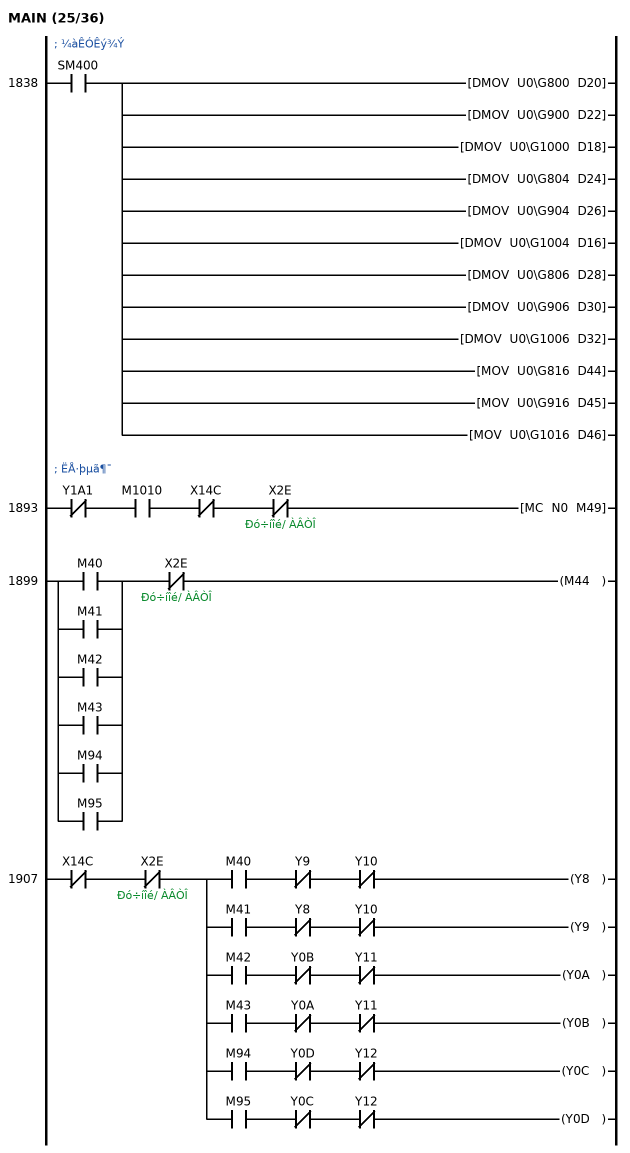
[picture p24: ladder of MAIN, rungs at steps 1838 to 1907]
; 监视数据
1838  LD      SM400
      DMOV    U0\G800 D20
      DMOV    U0\G900 D22
      DMOV    U0\G1000 D18
      DMOV    U0\G804 D24
      DMOV    U0\G904 D26
      DMOV    U0\G1004 D16
      DMOV    U0\G806 D28
      DMOV    U0\G906 D30
      DMOV    U0\G1006 D32
      MOV     U0\G816 D44
      MOV     U0\G916 D45
      MOV     U0\G1016 D46
; 伺服点动
1893  LDI     Y1A1
      AND     M1010
      ANI     X14C
      ANI     X2E  ; Ручной/ АВТО
      MC      N0 M49
1899  LD      M40
      OR      M41
      OR      M42
      OR      M43
      OR      M94
      OR      M95
      ANI     X2E  ; Ручной/ АВТО
      OUT     M44
1907  LDI     X14C
      ANI     X2E  ; Ручной/ АВТО
      MPS
      AND     M40
      ANI     Y9
      ANI     Y10
      OUT     Y8
      MRD
      AND     M41
      ANI     Y8
      ANI     Y10
      OUT     Y9
      MRD
      AND     M42
      ANI     Y0B
      ANI     Y11
      OUT     Y0A
      MRD
      AND     M43
      ANI     Y0A
      ANI     Y11
      OUT     Y0B
      MRD
      AND     M94
      ANI     Y0D
      ANI     Y12
      OUT     Y0C
      MPP
      AND     M95
      ANI     Y0C
      ANI     Y12
      OUT     Y0D
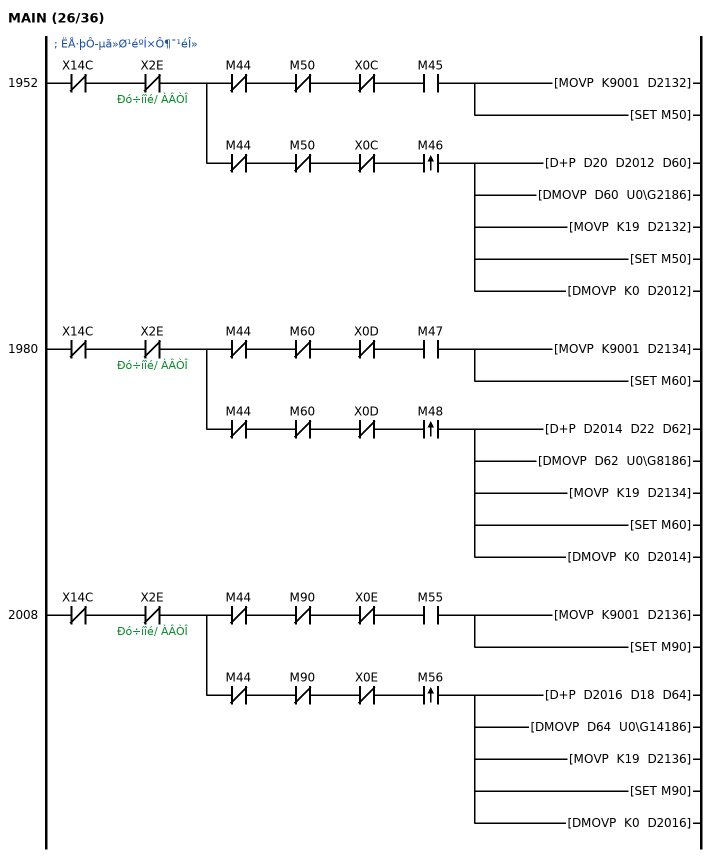
; 伺服原点回归和自动归位
1952  LDI     X14C
      ANI     X2E  ; Ручной/ АВТО
      MPS
      ANI     M44
      ANI     M50
      ANI     X0C
      AND     M45
      MOVP    K9001 D2132
      SET     M50
      MPP
      ANI     M44
      ANI     M50
      ANI     X0C
      ANDP    M46
      D+P     D20 D2012 D60
      DMOVP   D60 U0\G2186
      MOVP    K19 D2132
      SET     M50
      DMOVP   K0 D2012
1980  LDI     X14C
      ANI     X2E  ; Ручной/ АВТО
      MPS
      ANI     M44
      ANI     M60
      ANI     X0D
      AND     M47
      MOVP    K9001 D2134
      SET     M60
      MPP
      ANI     M44
      ANI     M60
      ANI     X0D
      ANDP    M48
      D+P     D2014 D22 D62
      DMOVP   D62 U0\G8186
      MOVP    K19 D2134
      SET     M60
      DMOVP   K0 D2014
2008  LDI     X14C
      ANI     X2E  ; Ручной/ АВТО
      MPS
      ANI     M44
      ANI     M90
      ANI     X0E
      AND     M55
      MOVP    K9001 D2136
      SET     M90
      MPP
      ANI     M44
      ANI     M90
      ANI     X0E
      ANDP    M56
      D+P     D2016 D18 D64
      DMOVP   D64 U0\G14186
      MOVP    K19 D2136
      SET     M90
      DMOVP   K0 D2016
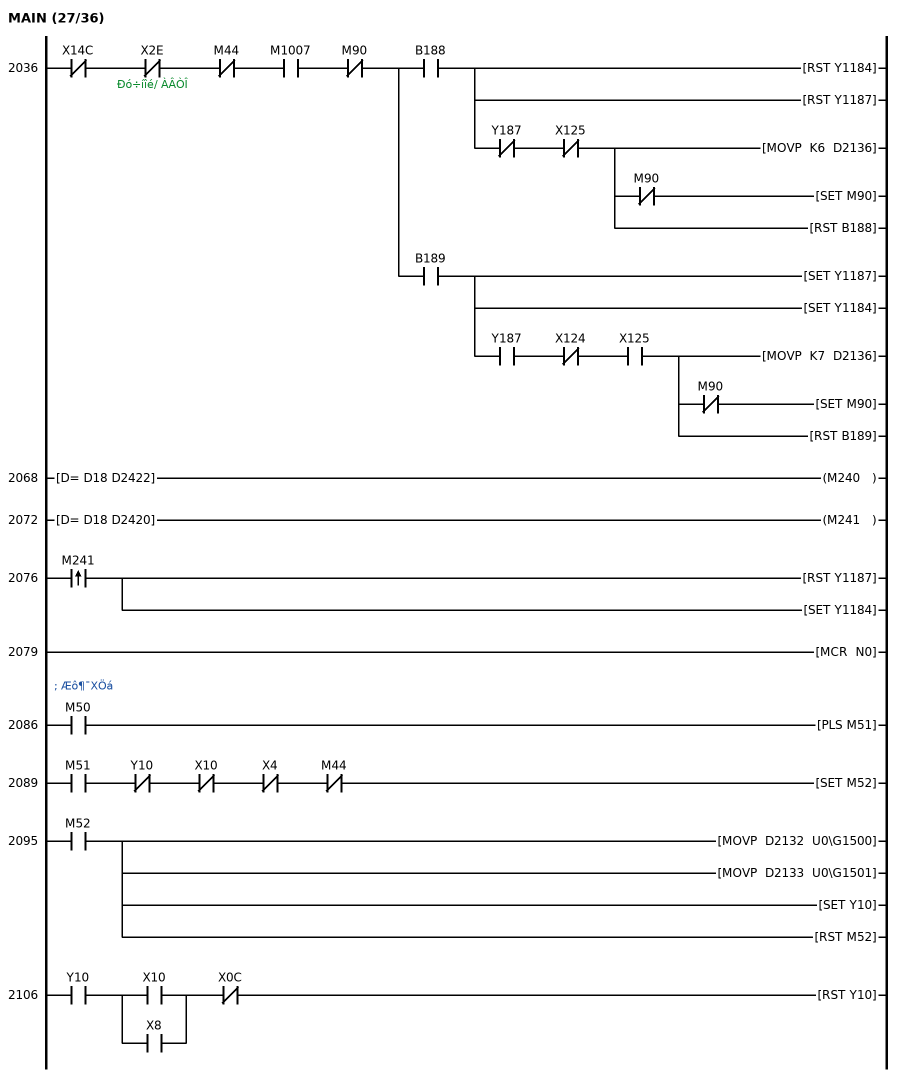
2036  LDI     X14C
      ANI     X2E  ; Ручной/ АВТО
      ANI     M44
      AND     M1007
      ANI     M90
      MPS
      AND     B188
      RST     Y1184
      RST     Y1187
      ANI     Y187
      ANI     X125
      MOVP    K6 D2136
      MPS
      ANI     M90
      SET     M90
      MPP
      RST     B188
      MPP
      AND     B189
      SET     Y1187
      SET     Y1184
      AND     Y187
      ANI     X124
      AND     X125
      MOVP    K7 D2136
      MPS
      ANI     M90
      SET     M90
      MPP
      RST     B189
2068  LDD=    D18 D2422
      OUT     M240
2072  LDD=    D18 D2420
      OUT     M241
2076  LDP     M241
      RST     Y1187
      SET     Y1184
2079  MCR     N0
; Æô¶¯XÖá
2086  LD      M50
      PLS     M51
2089  LD      M51
      ANI     Y10
      ANI     X10
      ANI     X4
      ANI     M44
      SET     M52
2095  LD      M52
      MOVP    D2132 U0\G1500
      MOVP    D2133 U0\G1501
      SET     Y10
      RST     M52
2106  LD      Y10
      LD      X10
      OR      X8
      ANB
      ANI     X0C
      RST     Y10
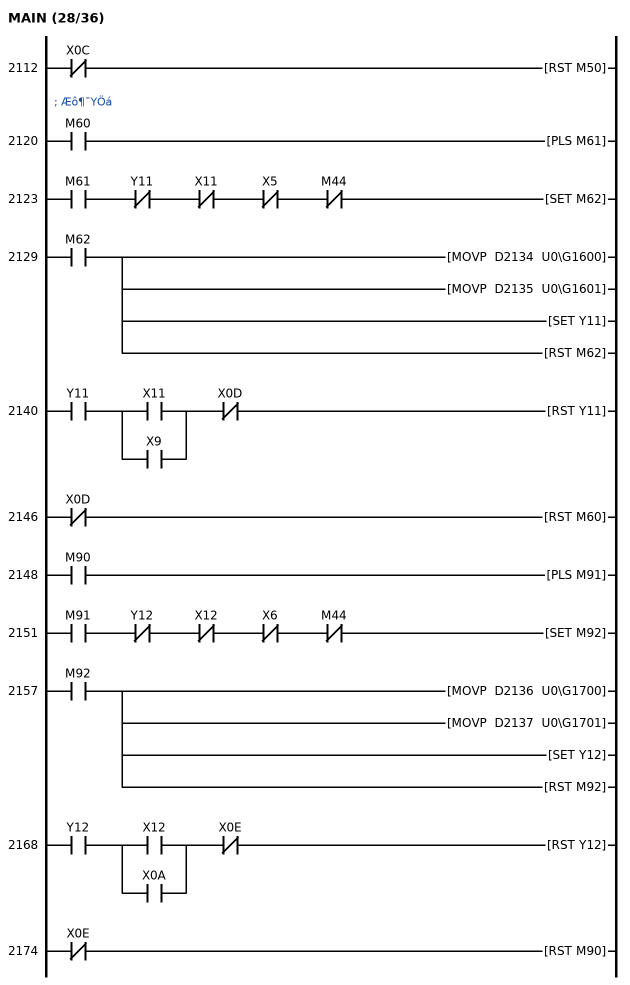
2112  LDI     X0C
      RST     M50
; Æô¶¯YÖá
2120  LD      M60
      PLS     M61
2123  LD      M61
      ANI     Y11
      ANI     X11
      ANI     X5
      ANI     M44
      SET     M62
2129  LD      M62
      MOVP    D2134 U0\G1600
      MOVP    D2135 U0\G1601
      SET     Y11
      RST     M62
2140  LD      Y11
      LD      X11
      OR      X9
      ANB
      ANI     X0D
      RST     Y11
2146  LDI     X0D
      RST     M60
2148  LD      M90
      PLS     M91
2151  LD      M91
      ANI     Y12
      ANI     X12
      ANI     X6
      ANI     M44
      SET     M92
2157  LD      M92
      MOVP    D2136 U0\G1700
      MOVP    D2137 U0\G1701
      SET     Y12
      RST     M92
2168  LD      Y12
      LD      X12
      OR      X0A
      ANB
      ANI     X0E
      RST     Y12
2174  LDI     X0E
      RST     M90
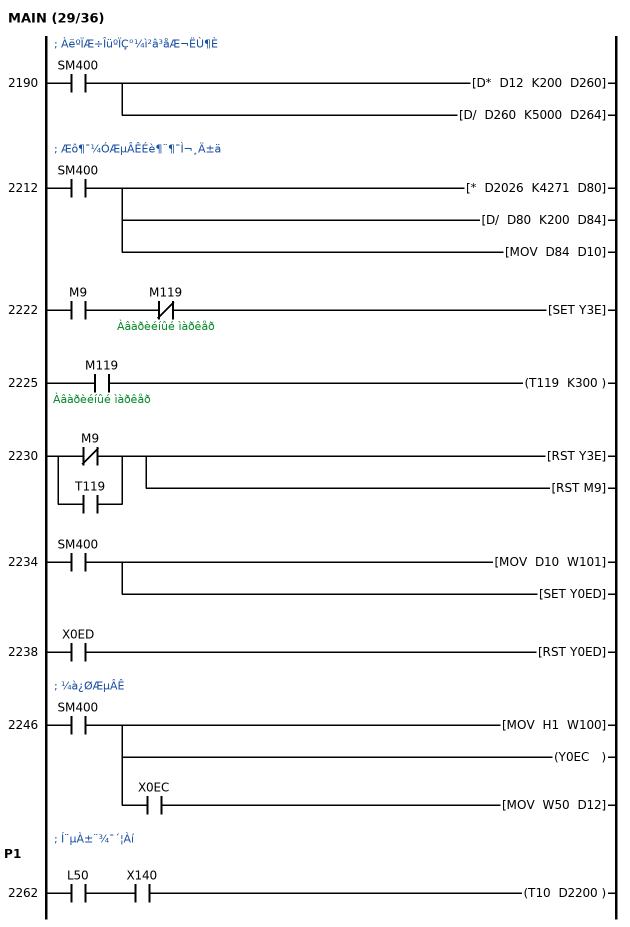
; 离合器吸合前检测冲片速度
2190  LD      SM400
      D*      D12 K200 D260
      D/      D260 K5000 D264
; 启动加频率设定动态改变
2212  LD      SM400
      *       D2026 K4271 D80
      D/      D80 K200 D84
      MOV     D84 D10
2222  LD      M9
      ANI     M119  ; Аварийный маркер
      SET     Y3E
2225  LD      M119  ; Аварийный маркер
      OUT     T119 K300
2230  LDI     M9
      OR      T119
      RST     Y3E
      RST     M9
2234  LD      SM400
      MOV     D10 W101
      SET     Y0ED
2238  LD      X0ED
      RST     Y0ED
; 监控频率
2246  LD      SM400
      MOV     H1 W100
      OUT     Y0EC
      AND     X0EC
      MOV     W50 D12
; 通道报警处理
      P1
2262  LD      L50
      AND     X140
      OUTH    T10 D2200
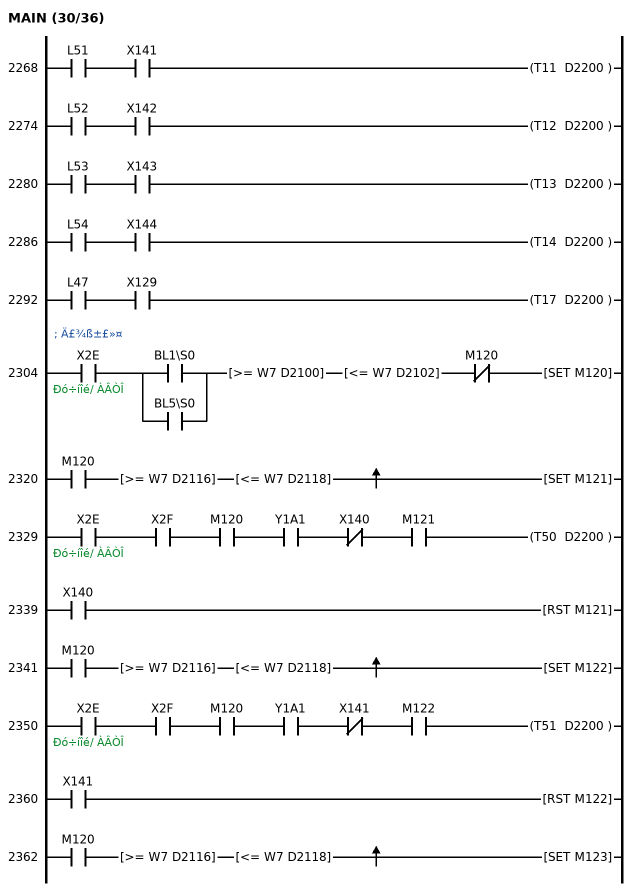
2268  LD      L51
      AND     X141
      OUTH    T11 D2200
2274  LD      L52
      AND     X142
      OUTH    T12 D2200
2280  LD      L53
      AND     X143
      OUTH    T13 D2200
2286  LD      L54
      AND     X144
      OUTH    T14 D2200
2292  LD      L47
      AND     X129
      OUTH    T17 D2200
; 模具保护
2304  LD      X2E  ; Ручной/ АВТО
      LD      BL1\S0
      OR      BL5\S0
      ANB
      AND>=   W7 D2100
      AND<=   W7 D2102
      ANI     M120
      SET     M120
2320  LD      M120
      AND>=   W7 D2116
      AND<=   W7 D2118
      MEP
      SET     M121
2329  LD      X2E  ; Ручной/ АВТО
      AND     X2F
      AND     M120
      AND     Y1A1
      ANI     X140
      AND     M121
      OUTH    T50 D2200
2339  LD      X140
      RST     M121
2341  LD      M120
      AND>=   W7 D2116
      AND<=   W7 D2118
      MEP
      SET     M122
2350  LD      X2E  ; Ручной/ АВТО
      AND     X2F
      AND     M120
      AND     Y1A1
      ANI     X141
      AND     M122
      OUTH    T51 D2200
2360  LD      X141
      RST     M122
2362  LD      M120
      AND>=   W7 D2116
      AND<=   W7 D2118
      MEP
      SET     M123
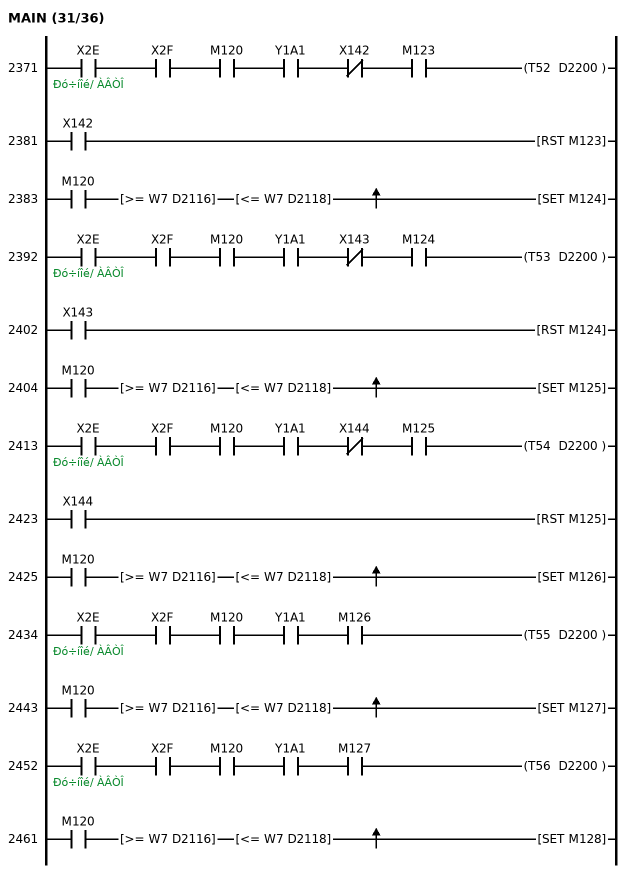
2371  LD      X2E  ; Ручной/ АВТО
      AND     X2F
      AND     M120
      AND     Y1A1
      ANI     X142
      AND     M123
      OUTH    T52 D2200
2381  LD      X142
      RST     M123
2383  LD      M120
      AND>=   W7 D2116
      AND<=   W7 D2118
      MEP
      SET     M124
2392  LD      X2E  ; Ручной/ АВТО
      AND     X2F
      AND     M120
      AND     Y1A1
      ANI     X143
      AND     M124
      OUTH    T53 D2200
2402  LD      X143
      RST     M124
2404  LD      M120
      AND>=   W7 D2116
      AND<=   W7 D2118
      MEP
      SET     M125
2413  LD      X2E  ; Ручной/ АВТО
      AND     X2F
      AND     M120
      AND     Y1A1
      ANI     X144
      AND     M125
      OUTH    T54 D2200
2423  LD      X144
      RST     M125
2425  LD      M120
      AND>=   W7 D2116
      AND<=   W7 D2118
      MEP
      SET     M126
2434  LD      X2E  ; Ручной/ АВТО
      AND     X2F
      AND     M120
      AND     Y1A1
      AND     M126
      OUTH    T55 D2200
2443  LD      M120
      AND>=   W7 D2116
      AND<=   W7 D2118
      MEP
      SET     M127
2452  LD      X2E  ; Ручной/ АВТО
      AND     X2F
      AND     M120
      AND     Y1A1
      AND     M127
      OUTH    T56 D2200
2461  LD      M120
      AND>=   W7 D2116
      AND<=   W7 D2118
      MEP
      SET     M128
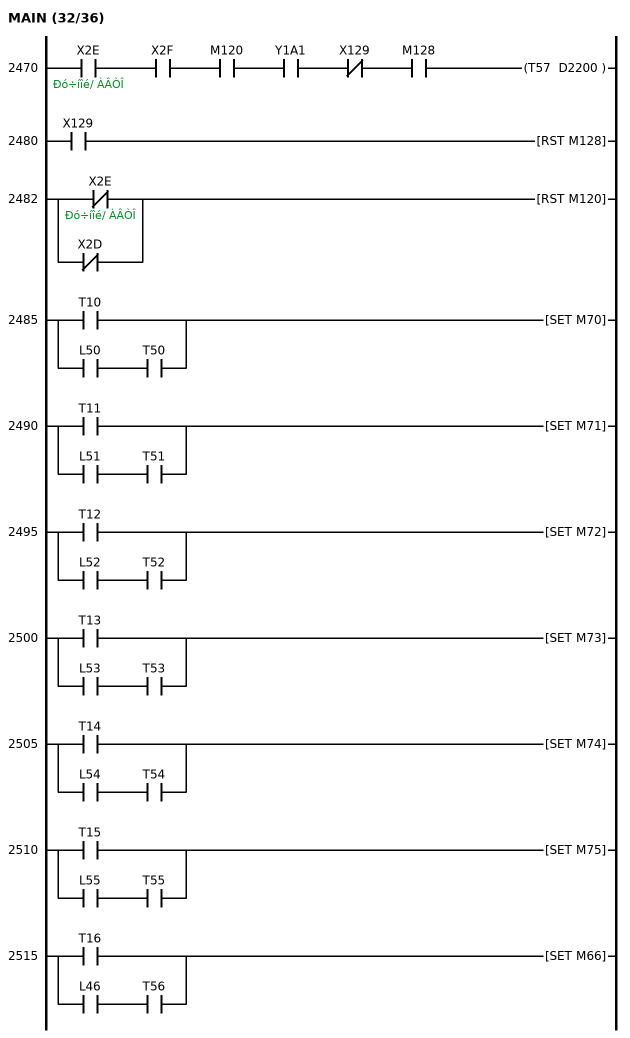
2470  LD      X2E  ; Ручной/ АВТО
      AND     X2F
      AND     M120
      AND     Y1A1
      ANI     X129
      AND     M128
      OUTH    T57 D2200
2480  LD      X129
      RST     M128
2482  LDI     X2E  ; Ручной/ АВТО
      ORI     X2D
      RST     M120
2485  LD      T10
      LD      L50
      AND     T50
      ORB
      SET     M70
2490  LD      T11
      LD      L51
      AND     T51
      ORB
      SET     M71
2495  LD      T12
      LD      L52
      AND     T52
      ORB
      SET     M72
2500  LD      T13
      LD      L53
      AND     T53
      ORB
      SET     M73
2505  LD      T14
      LD      L54
      AND     T54
      ORB
      SET     M74
2510  LD      T15
      LD      L55
      AND     T55
      ORB
      SET     M75
2515  LD      T16
      LD      L46
      AND     T56
      ORB
      SET     M66
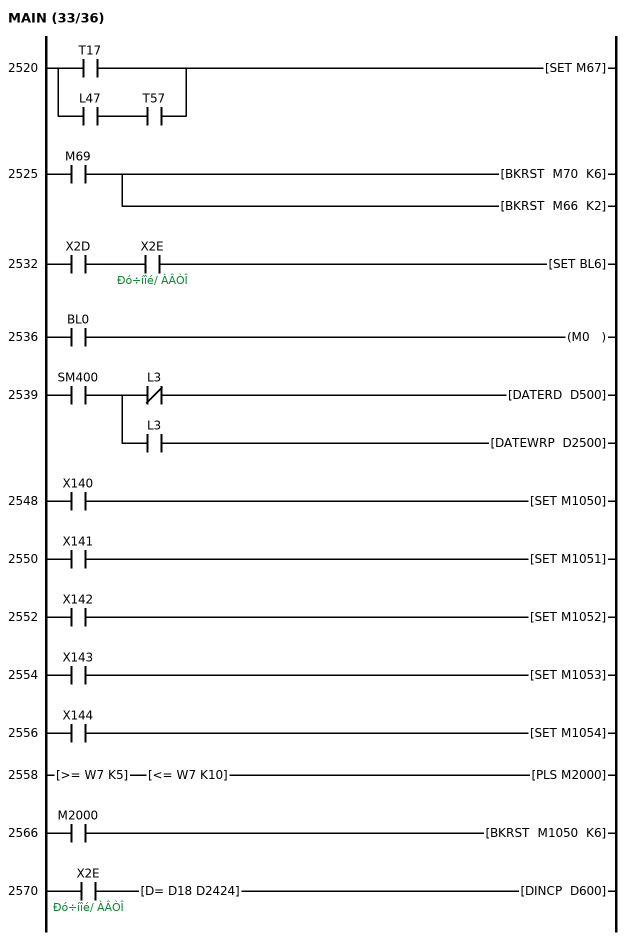
2520  LD      T17
      LD      L47
      AND     T57
      ORB
      SET     M67
2525  LD      M69
      BKRST   M70 K6
      BKRST   M66 K2
2532  LD      X2D
      AND     X2E  ; Ручной/ АВТО
      SET     BL6
2536  LD      BL0
      OUT     M0
2539  LD      SM400
      MPS
      ANI     L3
      DATERD  D500
      MPP
      AND     L3
      DATEWRP D2500
2548  LD      X140
      SET     M1050
2550  LD      X141
      SET     M1051
2552  LD      X142
      SET     M1052
2554  LD      X143
      SET     M1053
2556  LD      X144
      SET     M1054
2558  LD>=    W7 K5
      AND<=   W7 K10
      PLS     M2000
2566  LD      M2000
      BKRST   M1050 K6
2570  LD      X2E  ; Ручной/ АВТО
      ANDD=   D18 D2424
      DINCP   D600
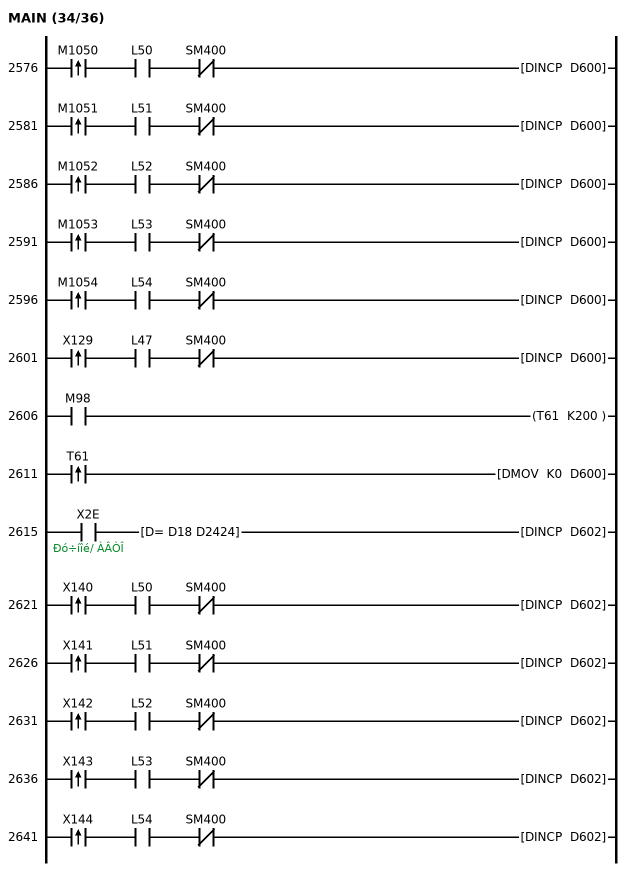
2576  LDP     M1050
      AND     L50
      ANI     SM400
      DINCP   D600
2581  LDP     M1051
      AND     L51
      ANI     SM400
      DINCP   D600
2586  LDP     M1052
      AND     L52
      ANI     SM400
      DINCP   D600
2591  LDP     M1053
      AND     L53
      ANI     SM400
      DINCP   D600
2596  LDP     M1054
      AND     L54
      ANI     SM400
      DINCP   D600
2601  LDP     X129
      AND     L47
      ANI     SM400
      DINCP   D600
2606  LD      M98
      OUT     T61 K200
2611  LDP     T61
      DMOV    K0 D600
2615  LD      X2E  ; Ручной/ АВТО
      ANDD=   D18 D2424
      DINCP   D602
2621  LDP     X140
      AND     L50
      ANI     SM400
      DINCP   D602
2626  LDP     X141
      AND     L51
      ANI     SM400
      DINCP   D602
2631  LDP     X142
      AND     L52
      ANI     SM400
      DINCP   D602
2636  LDP     X143
      AND     L53
      ANI     SM400
      DINCP   D602
2641  LDP     X144
      AND     L54
      ANI     SM400
      DINCP   D602
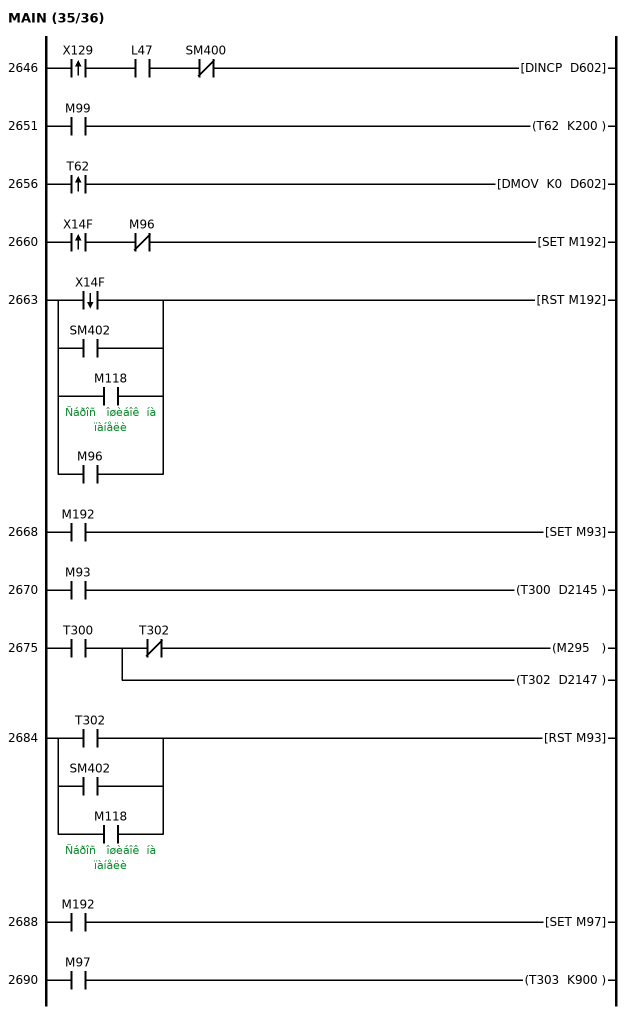
2646  LDP     X129
      AND     L47
      ANI     SM400
      DINCP   D602
2651  LD      M99
      OUT     T62 K200
2656  LDP     T62
      DMOV    K0 D602
2660  LDP     X14F
      ANI     M96
      SET     M192
2663  LDF     X14F
      OR      SM402
      OR      M118  ; Сброс   ошибок  на панели
      OR      M96
      RST     M192
2668  LD      M192
      SET     M93
2670  LD      M93
      OUTH    T300 D2145
2675  LD      T300
      MPS
      ANI     T302
      OUT     M295
      MPP
      OUTH    T302 D2147
2684  LD      T302
      OR      SM402
      OR      M118  ; Сброс   ошибок  на панели
      RST     M93
2688  LD      M192
      SET     M97
2690  LD      M97
      OUT     T303 K900
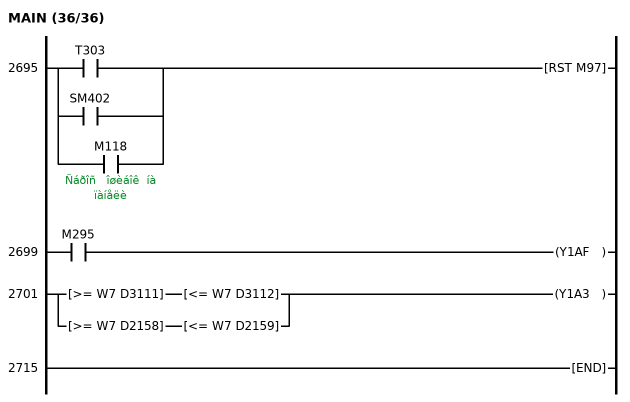
2695  LD      T303
      OR      SM402
      OR      M118  ; Сброс   ошибок  на панели
      RST     M97
2699  LD      M295
      OUT     Y1AF
2701  LD>=    W7 D3111
      AND<=   W7 D3112
      LD>=    W7 D2158
      AND<=   W7 D2159
      ORB
      OUT     Y1A3
2715  END
END_PROGRAM

// device comments not shown above
T131  ; Таймер2 выключения при  простое
